(* Logix 5000 project; controller Generic 1768-L43 rev 15.6; software revision 15.01; part 8 of 10 *)
(* tags used below, declared in another part *)
   AXIS_03 : AXIS_SERVO_DRIVE;
   Axis_03_CMD : UDT_Axis_CMD;
   Axis_03_Data : UDT_Axis_Data;
   Axis_03_MI : UDT_Motion_Instructions;
   Axis_03_Status : UDT_Axis_Status;
   AXIS_04 : AXIS_SERVO_DRIVE;
   Axis_04_CMD : UDT_Axis_CMD;
   Axis_04_Data : UDT_Axis_Data;
   Axis_04_MI : UDT_Motion_Instructions;
   Axis_04_Status : UDT_Axis_Status;
   GUI_RunSPD_NI : DINT;
   ManualControl : BOOL;
   MotionGroup : MOTION_GROUP;
   PowerUP_TMR : TIMER;
(* P03_AXIS_02, continued *)

ROUTINE R05_Manual   (* ladder *)
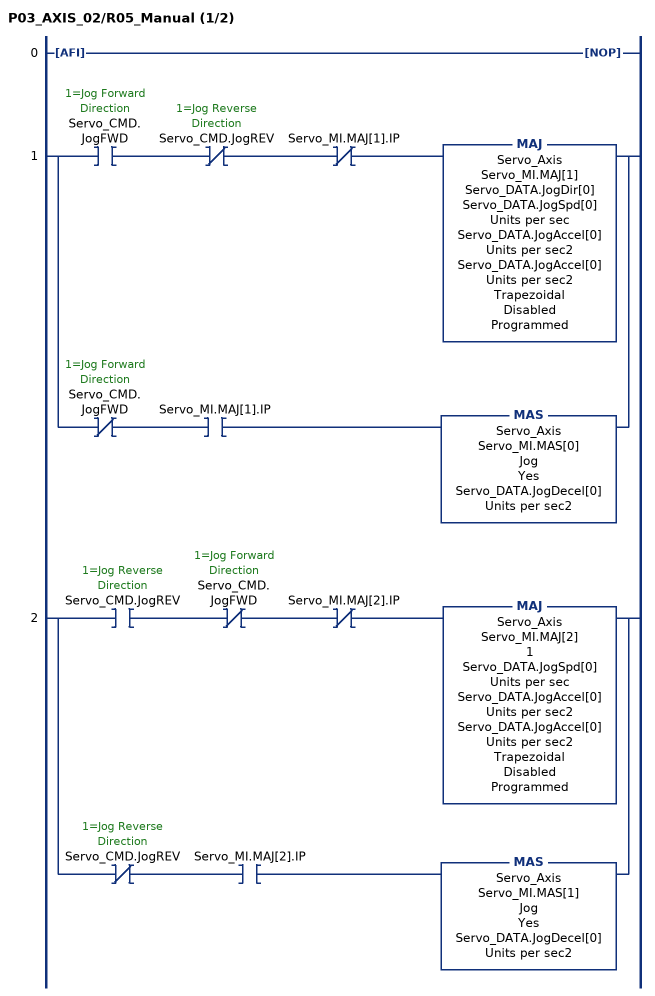
   0: AFI()NOP();
   1: [XIC(Servo_CMD.JogFWD) XIO(Servo_CMD.JogREV) XIO(Servo_MI.MAJ[1].IP) MAJ(Servo_Axis,Servo_MI.MAJ[1],Servo_DATA.JogDir[0],Servo_DATA.JogSpd[0],Units per sec,Servo_DATA.JogAccel[0],Units per sec2,Servo_DATA.JogAccel[0],Units per sec2,Trapezoidal,Disabled,Programmed) ,XIO(Servo_CMD.JogFWD) XIC(Servo_MI.MAJ[1].IP) MAS(Servo_Axis,Servo_MI.MAS[0],Jog,Yes,Servo_DATA.JogDecel[0],Units per sec2) ];
   2: [XIC(Servo_CMD.JogREV) XIO(Servo_CMD.JogFWD) XIO(Servo_MI.MAJ[2].IP) MAJ(Servo_Axis,Servo_MI.MAJ[2],1,Servo_DATA.JogSpd[0],Units per sec,Servo_DATA.JogAccel[0],Units per sec2,Servo_DATA.JogAccel[0],Units per sec2,Trapezoidal,Disabled,Programmed) ,XIO(Servo_CMD.JogREV) XIC(Servo_MI.MAJ[2].IP) MAS(Servo_Axis,Servo_MI.MAS[1],Jog,Yes,Servo_DATA.JogDecel[0],Units per sec2) ];
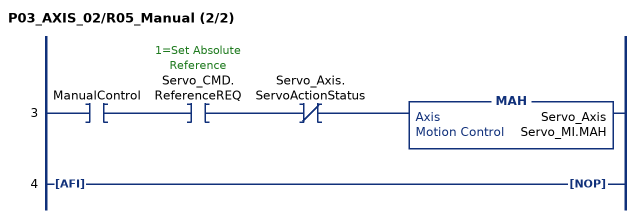
   3: XIC(ManualControl)XIC(Servo_CMD.ReferenceREQ)XIO(Servo_Axis.ServoActionStatus)MAH(Servo_Axis,Servo_MI.MAH);
   4: AFI()NOP();
END_ROUTINE

ROUTINE R06_AutoMotion   (* ladder *)
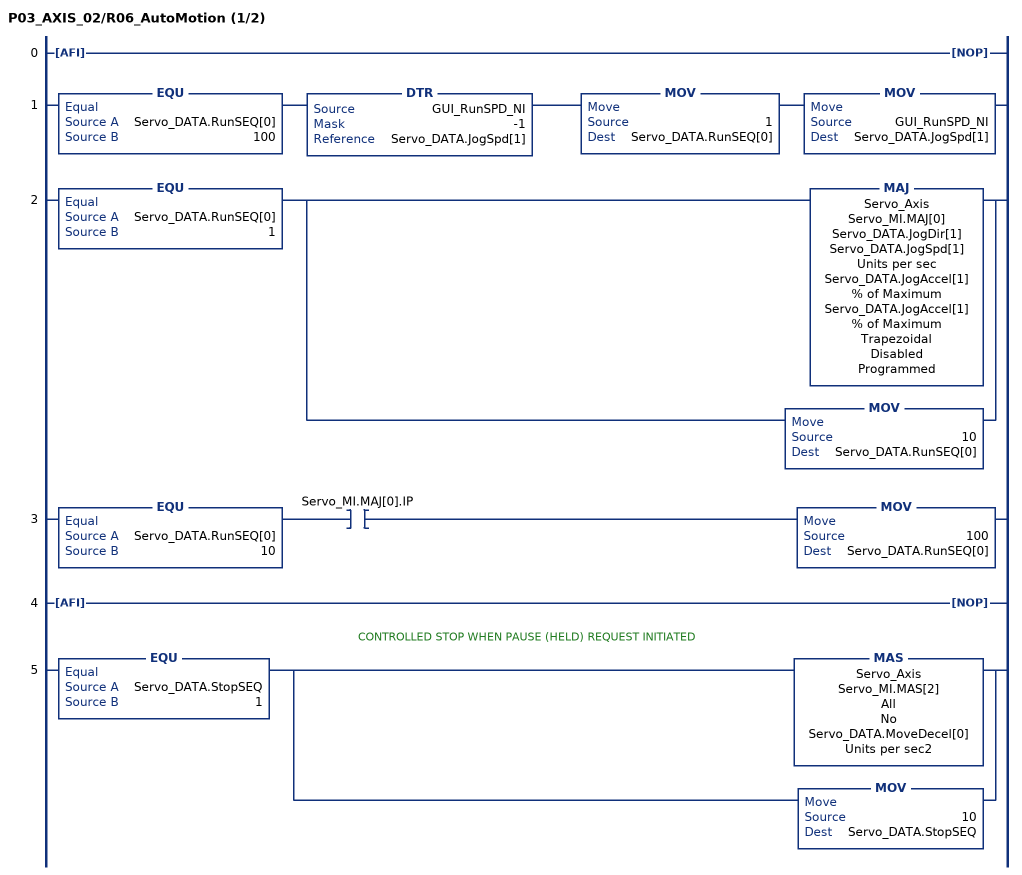
   0: AFI()NOP();
   1: EQU(Servo_DATA.RunSEQ[0],100)DTR(GUI_RunSPD_NI,-1,Servo_DATA.JogSpd[1])MOV(1,Servo_DATA.RunSEQ[0])MOV(GUI_RunSPD_NI,Servo_DATA.JogSpd[1]);
   2: EQU(Servo_DATA.RunSEQ[0],1)[MAJ(Servo_Axis,Servo_MI.MAJ[0],Servo_DATA.JogDir[1],Servo_DATA.JogSpd[1],Units per sec,Servo_DATA.JogAccel[1],% of Maximum,Servo_DATA.JogAccel[1],% of Maximum,Trapezoidal,Disabled,Programmed) ,MOV(10,Servo_DATA.RunSEQ[0]) ];
   3: EQU(Servo_DATA.RunSEQ[0],10)XIC(Servo_MI.MAJ[0].IP)MOV(100,Servo_DATA.RunSEQ[0]);
   4: AFI()NOP();
   // CONTROLLED STOP WHEN PAUSE (HELD) REQUEST INITIATED
   5: EQU(Servo_DATA.StopSEQ,1)[MAS(Servo_Axis,Servo_MI.MAS[2],All,No,Servo_DATA.MoveDecel[0],Units per sec2) ,MOV(10,Servo_DATA.StopSEQ) ];
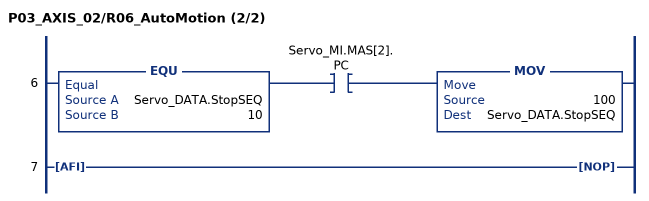
   6: EQU(Servo_DATA.StopSEQ,10)XIC(Servo_MI.MAS[2].PC)MOV(100,Servo_DATA.StopSEQ);
   7: AFI()NOP();
END_ROUTINE
END_PROGRAM

PROGRAM P04_AXIS_03   (* main routine R00_Dispatch *)
VAR
   Motion_Groups : ALIAS FOR MotionGroup;
   Servo_Axis : ALIAS FOR AXIS_03;
   Servo_CMD : ALIAS FOR Axis_03_CMD;
   Servo_DATA : ALIAS FOR Axis_03_Data;
   Servo_MI : ALIAS FOR Axis_03_MI;
   Servo_STATUS : ALIAS FOR Axis_03_Status;
END_VAR

ROUTINE R00_Dispatch   (* ladder *)
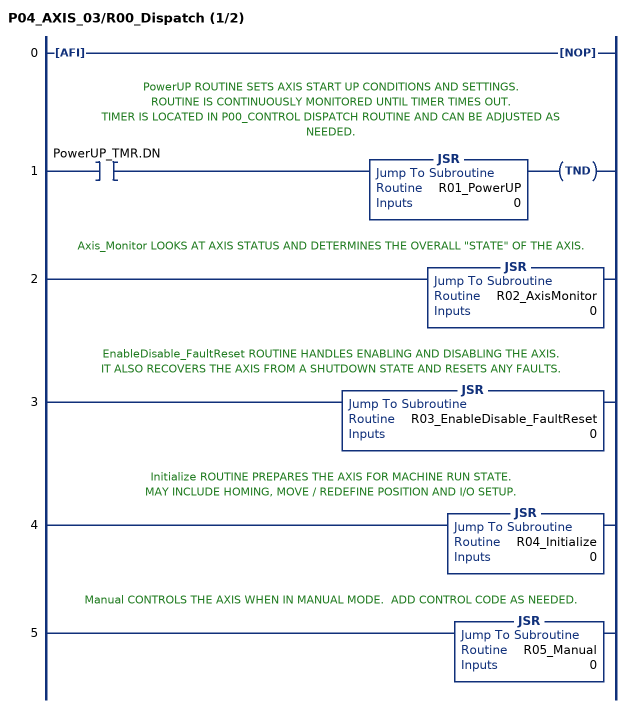
   0: AFI()NOP();
   // PowerUP ROUTINE SETS AXIS START UP CONDITIONS AND SETTINGS.
   // ROUTINE IS CONTINUOUSLY MONITORED UNTIL TIMER TIMES OUT.
   // TIMER IS LOCATED IN P00_CONTROL DISPATCH ROUTINE AND CAN BE ADJUSTED AS NEEDED.
   1: XIC(PowerUP_TMR.DN)JSR(R01_PowerUP,0)TND();
   // Axis_Monitor LOOKS AT AXIS STATUS AND DETERMINES THE OVERALL "STATE" OF THE AXIS.
   2: JSR(R02_AxisMonitor,0);
   // EnableDisable_FaultReset ROUTINE HANDLES ENABLING AND DISABLING THE AXIS.
   // IT ALSO RECOVERS THE AXIS FROM A SHUTDOWN STATE AND RESETS ANY FAULTS.
   3: JSR(R03_EnableDisable_FaultReset,0);
   // Initialize ROUTINE PREPARES THE AXIS FOR MACHINE RUN STATE.
   // MAY INCLUDE HOMING, MOVE / REDEFINE POSITION AND I/O SETUP.
   4: JSR(R04_Initialize,0);
   // Manual CONTROLS THE AXIS WHEN IN MANUAL MODE.  ADD CONTROL CODE AS NEEDED.
   5: JSR(R05_Manual,0);
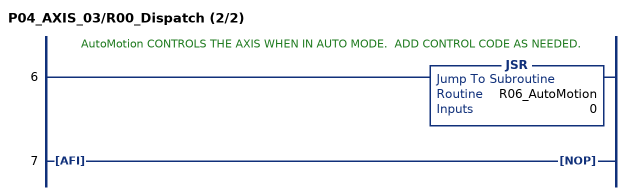
   // AutoMotion CONTROLS THE AXIS WHEN IN AUTO MODE.  ADD CONTROL CODE AS NEEDED.
   6: JSR(R06_AutoMotion,0);
   7: AFI()NOP();
END_ROUTINE

ROUTINE R01_PowerUP   (* ladder *)
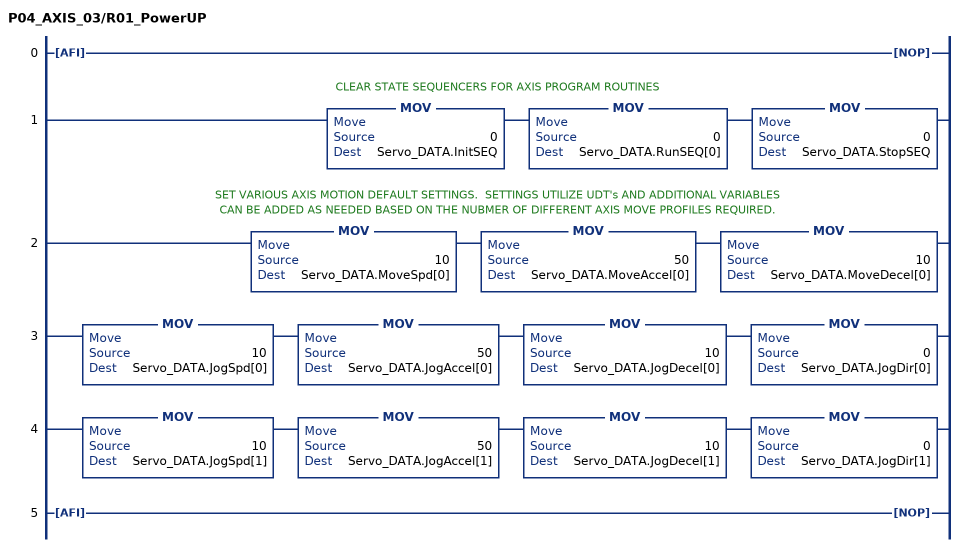
   0: AFI()NOP();
   // CLEAR STATE SEQUENCERS FOR AXIS PROGRAM ROUTINES
   1: MOV(0,Servo_DATA.InitSEQ)MOV(0,Servo_DATA.RunSEQ[0])MOV(0,Servo_DATA.StopSEQ);
   // SET VARIOUS AXIS MOTION DEFAULT SETTINGS.  SETTINGS UTILIZE UDT's AND ADDITIONAL VARIABLES
   // CAN BE ADDED AS NEEDED BASED ON THE NUBMER OF DIFFERENT AXIS MOVE PROFILES REQUIRED.
   2: MOV(10,Servo_DATA.MoveSpd[0])MOV(50,Servo_DATA.MoveAccel[0])MOV(10,Servo_DATA.MoveDecel[0]);
   3: MOV(10,Servo_DATA.JogSpd[0])MOV(50,Servo_DATA.JogAccel[0])MOV(10,Servo_DATA.JogDecel[0])MOV(0,Servo_DATA.JogDir[0]);
   4: MOV(10,Servo_DATA.JogSpd[1])MOV(50,Servo_DATA.JogAccel[1])MOV(10,Servo_DATA.JogDecel[1])MOV(0,Servo_DATA.JogDir[1]);
   5: AFI()NOP();
END_ROUTINE

ROUTINE R02_AxisMonitor   (* ladder *)
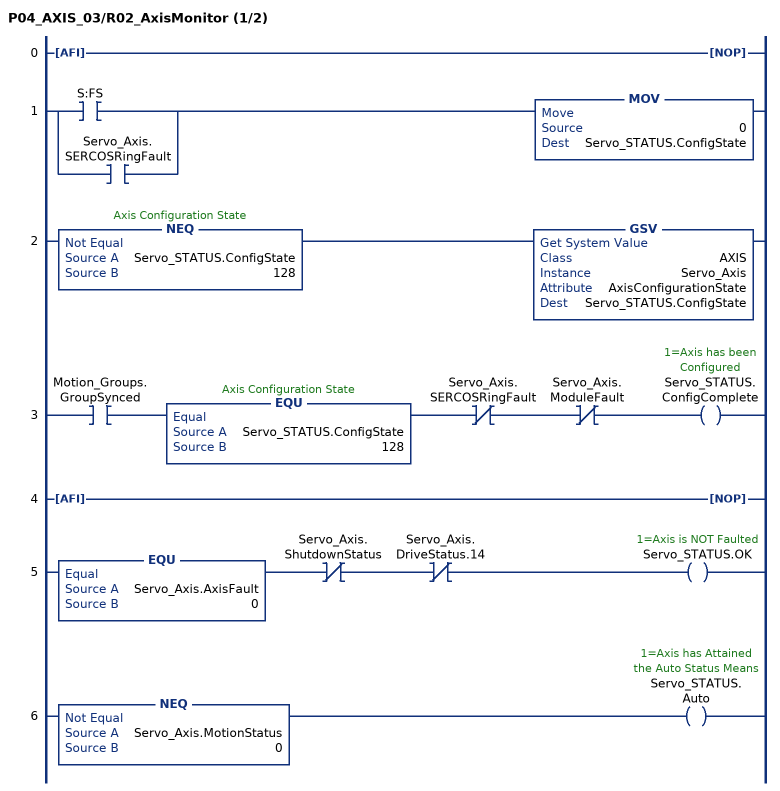
   0: AFI()NOP();
   1: [XIC(S:FS) ,XIC(Servo_Axis.SERCOSRingFault) ]MOV(0,Servo_STATUS.ConfigState);
   2: NEQ(Servo_STATUS.ConfigState,128)GSV(AXIS,Servo_Axis,AxisConfigurationState,Servo_STATUS.ConfigState);
   3: XIC(Motion_Groups.GroupSynced)EQU(Servo_STATUS.ConfigState,128)XIO(Servo_Axis.SERCOSRingFault)XIO(Servo_Axis.ModuleFault)OTE(Servo_STATUS.ConfigComplete);
   4: AFI()NOP();
   5: EQU(Servo_Axis.AxisFault,0)XIO(Servo_Axis.ShutdownStatus)XIO(Servo_Axis.DriveStatus.14)OTE(Servo_STATUS.OK);
   6: NEQ(Servo_Axis.MotionStatus,0)OTE(Servo_STATUS.Auto);
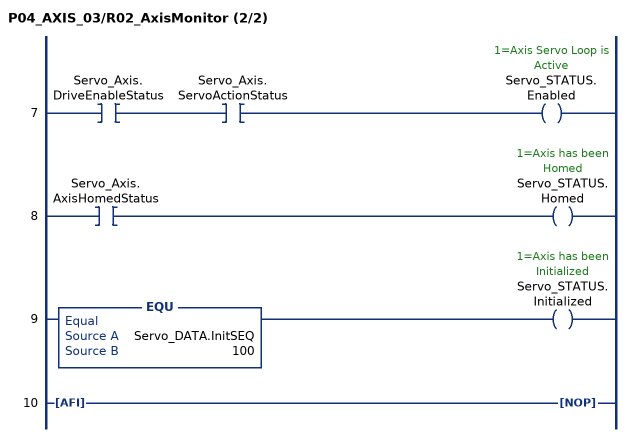
   7: XIC(Servo_Axis.DriveEnableStatus)XIC(Servo_Axis.ServoActionStatus)OTE(Servo_STATUS.Enabled);
   8: XIC(Servo_Axis.AxisHomedStatus)OTE(Servo_STATUS.Homed);
   9: EQU(Servo_DATA.InitSEQ,100)OTE(Servo_STATUS.Initialized);
   10: AFI()NOP();
END_ROUTINE

ROUTINE R03_EnableDisable_FaultReset   (* ladder *)
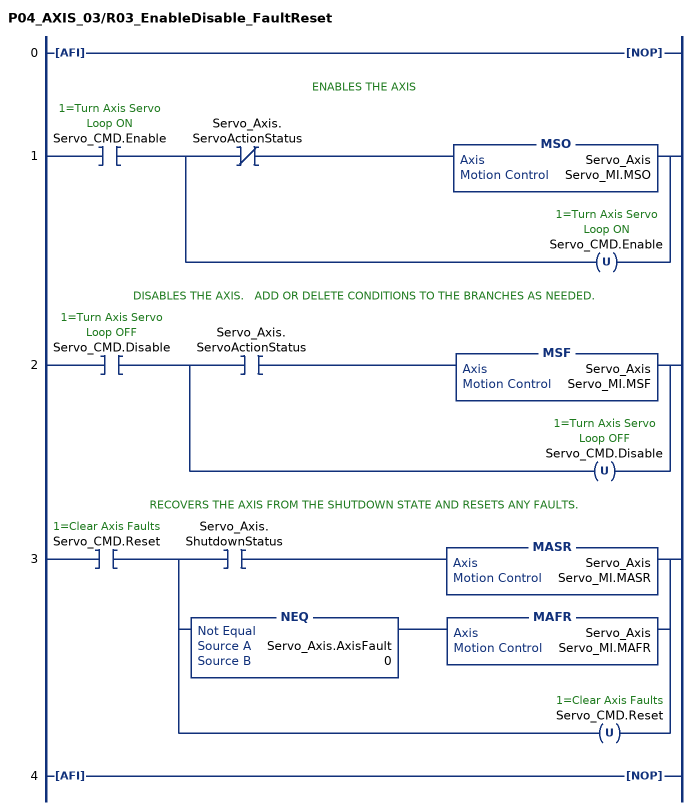
   0: AFI()NOP();
   // ENABLES THE AXIS
   1: XIC(Servo_CMD.Enable)[XIO(Servo_Axis.ServoActionStatus) MSO(Servo_Axis,Servo_MI.MSO) ,OTU(Servo_CMD.Enable) ];
   // DISABLES THE AXIS.   ADD OR DELETE CONDITIONS TO THE BRANCHES AS NEEDED.
   2: XIC(Servo_CMD.Disable)[XIC(Servo_Axis.ServoActionStatus) MSF(Servo_Axis,Servo_MI.MSF) ,OTU(Servo_CMD.Disable) ];
   // RECOVERS THE AXIS FROM THE SHUTDOWN STATE AND RESETS ANY FAULTS.
   3: XIC(Servo_CMD.Reset)[XIC(Servo_Axis.ShutdownStatus) MASR(Servo_Axis,Servo_MI.MASR) ,NEQ(Servo_Axis.AxisFault,0) MAFR(Servo_Axis,Servo_MI.MAFR) ,OTU(Servo_CMD.Reset) ];
   4: AFI()NOP();
END_ROUTINE

ROUTINE R04_Initialize   (* ladder *)
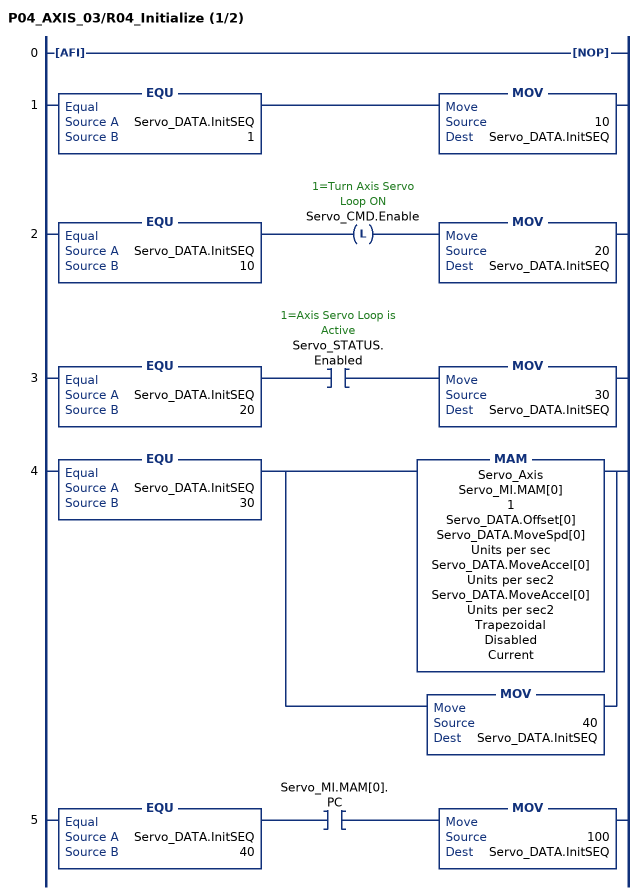
   0: AFI()NOP();
   1: EQU(Servo_DATA.InitSEQ,1)MOV(10,Servo_DATA.InitSEQ);
   2: EQU(Servo_DATA.InitSEQ,10)OTL(Servo_CMD.Enable)MOV(20,Servo_DATA.InitSEQ);
   3: EQU(Servo_DATA.InitSEQ,20)XIC(Servo_STATUS.Enabled)MOV(30,Servo_DATA.InitSEQ);
   4: EQU(Servo_DATA.InitSEQ,30)[MAM(Servo_Axis,Servo_MI.MAM[0],1,Servo_DATA.Offset[0],Servo_DATA.MoveSpd[0],Units per sec,Servo_DATA.MoveAccel[0],Units per sec2,Servo_DATA.MoveAccel[0],Units per sec2,Trapezoidal,Disabled,Current) ,MOV(40,Servo_DATA.InitSEQ) ];
   5: EQU(Servo_DATA.InitSEQ,40)XIC(Servo_MI.MAM[0].PC)MOV(100,Servo_DATA.InitSEQ);
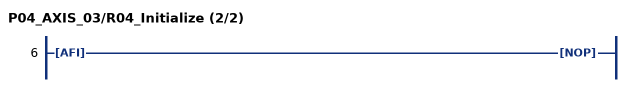
   6: AFI()NOP();
END_ROUTINE

ROUTINE R05_Manual   (* ladder *)
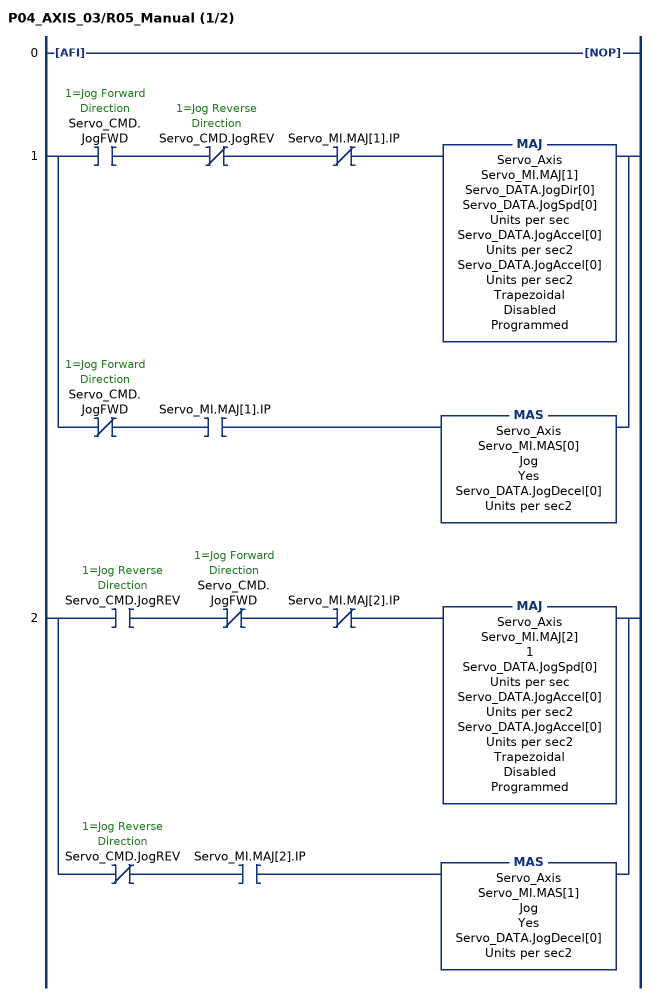
   0: AFI()NOP();
   1: [XIC(Servo_CMD.JogFWD) XIO(Servo_CMD.JogREV) XIO(Servo_MI.MAJ[1].IP) MAJ(Servo_Axis,Servo_MI.MAJ[1],Servo_DATA.JogDir[0],Servo_DATA.JogSpd[0],Units per sec,Servo_DATA.JogAccel[0],Units per sec2,Servo_DATA.JogAccel[0],Units per sec2,Trapezoidal,Disabled,Programmed) ,XIO(Servo_CMD.JogFWD) XIC(Servo_MI.MAJ[1].IP) MAS(Servo_Axis,Servo_MI.MAS[0],Jog,Yes,Servo_DATA.JogDecel[0],Units per sec2) ];
   2: [XIC(Servo_CMD.JogREV) XIO(Servo_CMD.JogFWD) XIO(Servo_MI.MAJ[2].IP) MAJ(Servo_Axis,Servo_MI.MAJ[2],1,Servo_DATA.JogSpd[0],Units per sec,Servo_DATA.JogAccel[0],Units per sec2,Servo_DATA.JogAccel[0],Units per sec2,Trapezoidal,Disabled,Programmed) ,XIO(Servo_CMD.JogREV) XIC(Servo_MI.MAJ[2].IP) MAS(Servo_Axis,Servo_MI.MAS[1],Jog,Yes,Servo_DATA.JogDecel[0],Units per sec2) ];
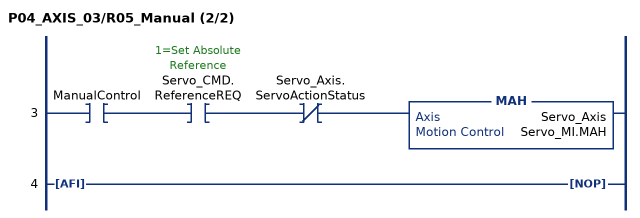
   3: XIC(ManualControl)XIC(Servo_CMD.ReferenceREQ)XIO(Servo_Axis.ServoActionStatus)MAH(Servo_Axis,Servo_MI.MAH);
   4: AFI()NOP();
END_ROUTINE

ROUTINE R06_AutoMotion   (* ladder *)
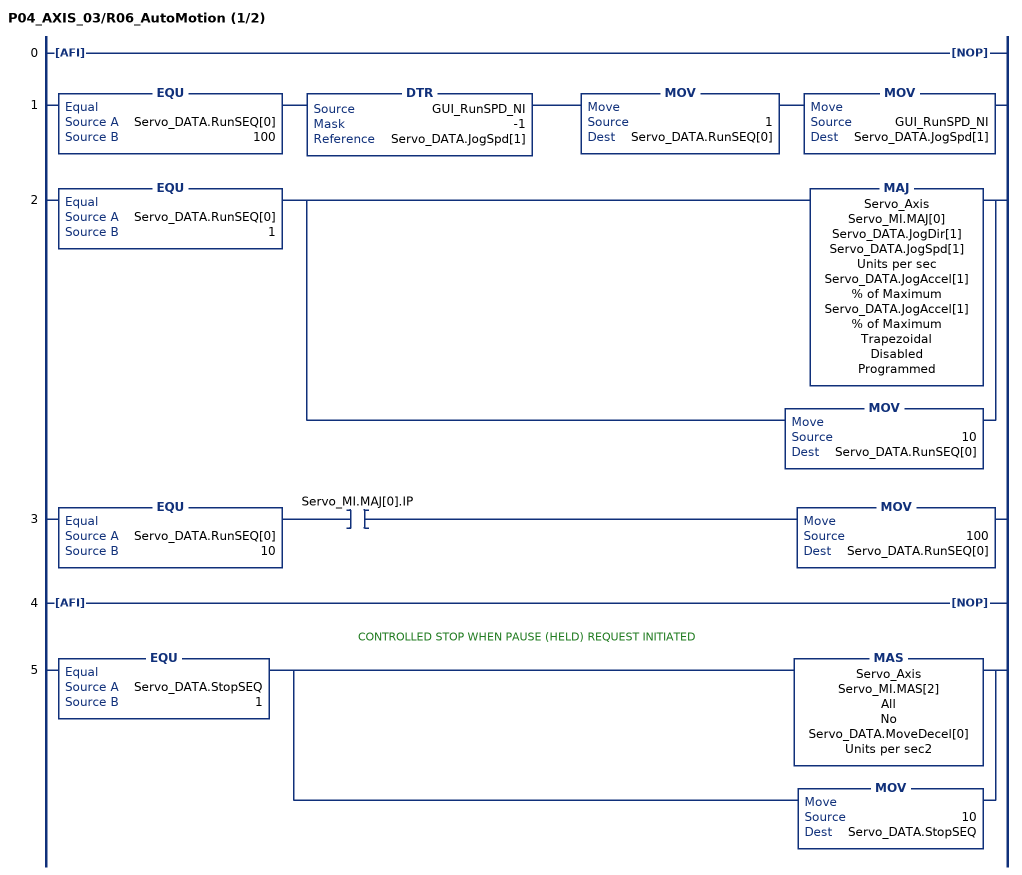
   0: AFI()NOP();
   1: EQU(Servo_DATA.RunSEQ[0],100)DTR(GUI_RunSPD_NI,-1,Servo_DATA.JogSpd[1])MOV(1,Servo_DATA.RunSEQ[0])MOV(GUI_RunSPD_NI,Servo_DATA.JogSpd[1]);
   2: EQU(Servo_DATA.RunSEQ[0],1)[MAJ(Servo_Axis,Servo_MI.MAJ[0],Servo_DATA.JogDir[1],Servo_DATA.JogSpd[1],Units per sec,Servo_DATA.JogAccel[1],% of Maximum,Servo_DATA.JogAccel[1],% of Maximum,Trapezoidal,Disabled,Programmed) ,MOV(10,Servo_DATA.RunSEQ[0]) ];
   3: EQU(Servo_DATA.RunSEQ[0],10)XIC(Servo_MI.MAJ[0].IP)MOV(100,Servo_DATA.RunSEQ[0]);
   4: AFI()NOP();
   // CONTROLLED STOP WHEN PAUSE (HELD) REQUEST INITIATED
   5: EQU(Servo_DATA.StopSEQ,1)[MAS(Servo_Axis,Servo_MI.MAS[2],All,No,Servo_DATA.MoveDecel[0],Units per sec2) ,MOV(10,Servo_DATA.StopSEQ) ];
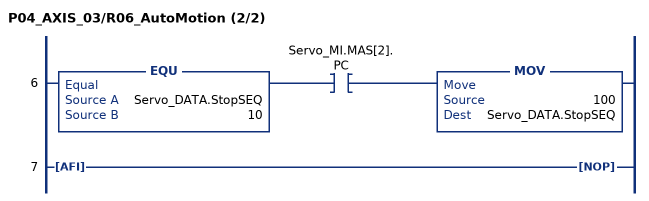
   6: EQU(Servo_DATA.StopSEQ,10)XIC(Servo_MI.MAS[2].PC)MOV(100,Servo_DATA.StopSEQ);
   7: AFI()NOP();
END_ROUTINE
END_PROGRAM

PROGRAM P05_AXIS_04   (* main routine R00_Dispatch *)
VAR
   Motion_Groups : ALIAS FOR MotionGroup;
   Servo_Axis : ALIAS FOR AXIS_04;
   Servo_CMD : ALIAS FOR Axis_04_CMD;
   Servo_DATA : ALIAS FOR Axis_04_Data;
   Servo_MI : ALIAS FOR Axis_04_MI;
   Servo_STATUS : ALIAS FOR Axis_04_Status;
END_VAR

ROUTINE R00_Dispatch   (* ladder *)
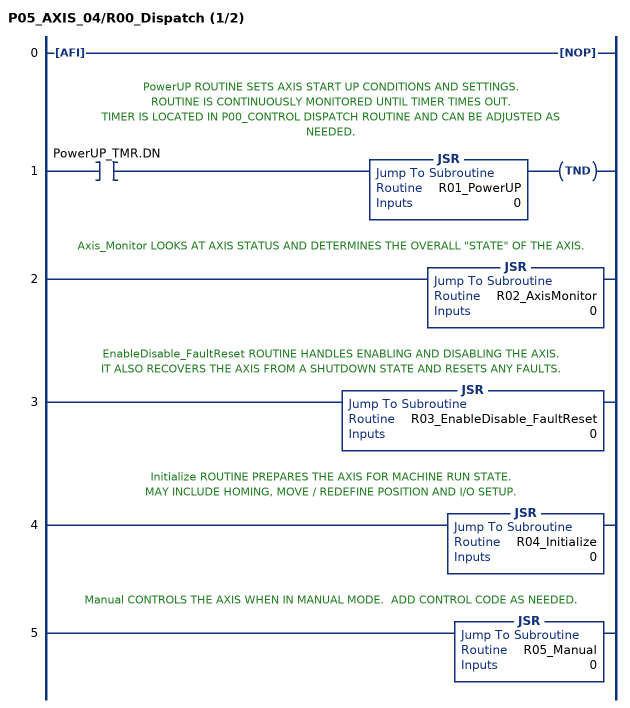
   0: AFI()NOP();
   // PowerUP ROUTINE SETS AXIS START UP CONDITIONS AND SETTINGS.
   // ROUTINE IS CONTINUOUSLY MONITORED UNTIL TIMER TIMES OUT.
   // TIMER IS LOCATED IN P00_CONTROL DISPATCH ROUTINE AND CAN BE ADJUSTED AS NEEDED.
   1: XIC(PowerUP_TMR.DN)JSR(R01_PowerUP,0)TND();
   // Axis_Monitor LOOKS AT AXIS STATUS AND DETERMINES THE OVERALL "STATE" OF THE AXIS.
   2: JSR(R02_AxisMonitor,0);
   // EnableDisable_FaultReset ROUTINE HANDLES ENABLING AND DISABLING THE AXIS.
   // IT ALSO RECOVERS THE AXIS FROM A SHUTDOWN STATE AND RESETS ANY FAULTS.
   3: JSR(R03_EnableDisable_FaultReset,0);
   // Initialize ROUTINE PREPARES THE AXIS FOR MACHINE RUN STATE.
   // MAY INCLUDE HOMING, MOVE / REDEFINE POSITION AND I/O SETUP.
   4: JSR(R04_Initialize,0);
   // Manual CONTROLS THE AXIS WHEN IN MANUAL MODE.  ADD CONTROL CODE AS NEEDED.
   5: JSR(R05_Manual,0);
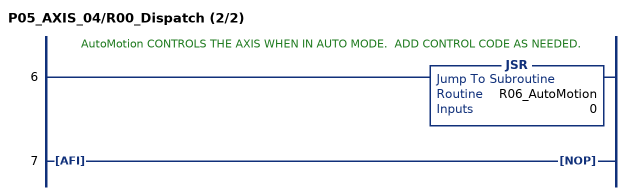
   // AutoMotion CONTROLS THE AXIS WHEN IN AUTO MODE.  ADD CONTROL CODE AS NEEDED.
   6: JSR(R06_AutoMotion,0);
   7: AFI()NOP();
END_ROUTINE
